TYPE ST_HMI_CONTROL_SETTING_STATION_OUT :
STRUCT
	stControlSetting	: ST_HMI_CONTROL_SETTING_ITEM_OUT;
	stSettingView		: ARRAY[0..CONST.iMaxIdxLocalSetting] OF ST_Data_Item_String;
END_STRUCT
END_TYPE

(* stored: Version 1.1.0.1, ProductVersion 3.1.4024.12
   DUT ST_HMI_CONTROL_SETTING_STATION_OUT: Id {b27c428c-8539-4129-ad15-dd0ee8d78e0c} *)
